// Mitsubishi GX Works2 project: mc연습   PLC: Q02/Q02H

PROGRAM MAIN
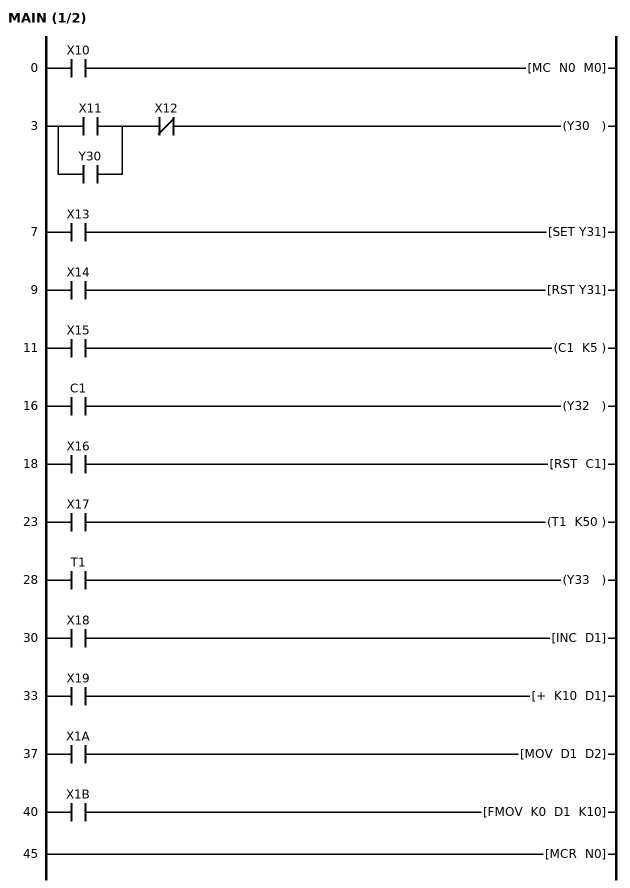
0     LD      X10
      MC      N0 M0
3     LD      X11
      OR      Y30
      ANI     X12
      OUT     Y30
7     LD      X13
      SET     Y31
9     LD      X14
      RST     Y31
11    LD      X15
      OUT     C1 K5
16    LD      C1
      OUT     Y32
18    LD      X16
      RST     C1
23    LD      X17
      OUT     T1 K50
28    LD      T1
      OUT     Y33
30    LD      X18
      INC     D1
33    LD      X19
      +       K10 D1
37    LD      X1A
      MOV     D1 D2
40    LD      X1B
      FMOV    K0 D1 K10
45    MCR     N0
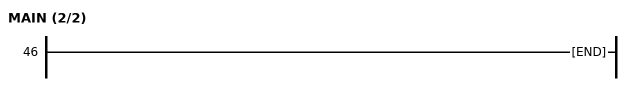
46    END
END_PROGRAM
